INTERFACE ITF_BaseFlagSet

METHOD PUBLIC SetFlag
VAR_INPUT
	bState				: BOOL;
END_VAR
END_METHOD

END_INTERFACE

(* stored: Version 1.1.0.1
   Itf ITF_BaseFlagSet: Id {adfc721f-2d18-0ae5-076c-500568af33b4}
   Method SetFlag: Id {468fe690-b436-00c7-2772-f4df5ee911d4} *)
